KUKA KRL program: pickpallet2.src, pickpallet2.dat

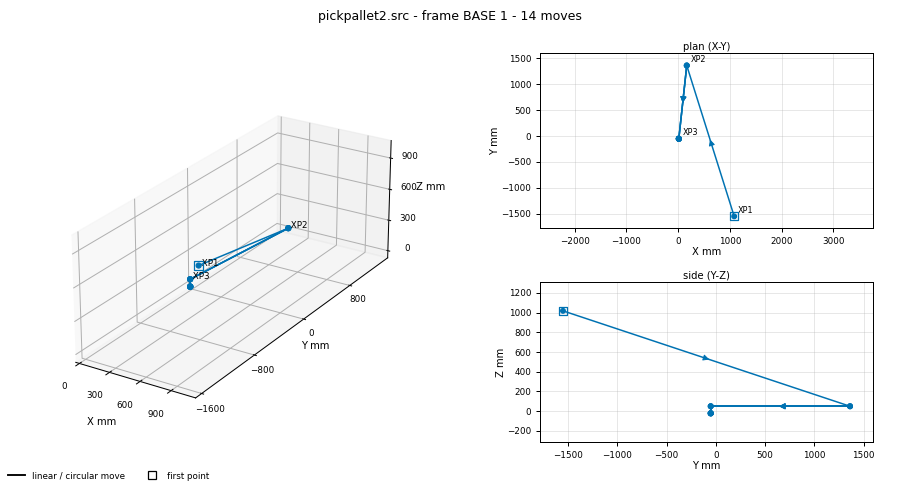
[picture p0: tool path of pickpallet2.src in frame BASE 1, 14 of 20 moves have a stored position in this frame; points joined in program order, loops and branches not executed]
--- pickpallet2.src ---
&ACCESS RVO1
&COMMENT
&ACCESS RVP
&PARAM EDITMASK = *
&PARAM TEMPLATE = C:\KRC\Roboter\Template\vorgabe
&PARAM DISKPATH = KRC:\R1\Program
DEF pickpallet2(pallet1_num:in, Z_pallet:in)
decl pos poz_vz_pal
decl int pallet1_num, ip, Z_pallet
DECL REAL low_z_pallet_pick
decl pos actual_pick_point_1, pallet_pick_point, prp1, prp2, prp9, prp4, prp5

low_z_pallet_pick = 20 ; mm, Z coordinate of the bottom of the first pallet at the pallet pick place

; rotation to the pallet pick place
;FOLD PTP P1  Vel=100 % PDAT1 Tool[2]:tool_empty Base[1]:PickPallet1;%{PE}%R 8.3.22,%MKUKATPBASIS,%CMOVE,%VPTP,%P 1:PTP, 2:P1, 3:, 5:100, 7:PDAT1
$BWDSTART=FALSE
PDAT_ACT=PPDAT1
FDAT_ACT=FP1
BAS(#PTP_PARAMS,100)
PTP XP1
;ENDFOLD

if ((pallet1_num == 10) or (FLAG[5] == FALSE)) then
; movement to the top with search

; rising up
;FOLD LIN P2  Vel=2.00000 m/s CPDAT2 Tool[2]:tool_empty Base[1]:PickPallet1;%{PE}%R 8.3.22,%MKUKATPBASIS,%CMOVE,%VLIN,%P 1:LIN, 2:P2, 3:, 5:2.00000, 7:CPDAT2
$BWDSTART=FALSE
LDAT_ACT=LCPDAT2
FDAT_ACT=FP2
BAS(#CP_PARAMS,2.00000)
LIN XP2
;ENDFOLD

; taking air in order not to avoid the hooks opening
;FOLD SYN OUT 1 'Finger_right'  State= TRUE  at END  Delay= 1500 ms;%{PE}%R 8.3.22,%MKUKATPBASIS,%COUT,%VSYNOUT,%P 2:1, 3:Finger_right, 5:TRUE, 7:1, 9:0, 12:1500
TRIGGER WHEN DISTANCE=1 DELAY=1500 DO $OUT[1]=TRUE
;ENDFOLD
;FOLD SYN OUT 3 'Finger_left'  State= TRUE  at START  Delay= 1500 ms;%{PE}%R 8.3.22,%MKUKATPBASIS,%COUT,%VSYNOUT,%P 2:3, 3:Finger_left, 5:TRUE, 7:0, 9:0, 12:1500
TRIGGER WHEN DISTANCE=0 DELAY=1500 DO $OUT[3]=TRUE
;ENDFOLD

; opening the hooks
;FOLD SYN OUT 5 'All_hooks'  State= TRUE  at END  Delay= 500 ms;%{PE}%R 8.3.22,%MKUKATPBASIS,%COUT,%VSYNOUT,%P 2:5, 3:All_hooks, 5:TRUE, 7:1, 9:0, 12:500
TRIGGER WHEN DISTANCE=1 DELAY=500 DO $OUT[5]=TRUE
;ENDFOLD

; moving to the point above pallet pick place
;FOLD LIN P3  Vel=2.00000 m/s CPDAT3 Tool[2]:tool_empty Base[1]:PickPallet1;%{PE}%R 8.3.22,%MKUKATPBASIS,%CMOVE,%VLIN,%P 1:LIN, 2:P3, 3:, 5:2.00000, 7:CPDAT3
$BWDSTART=FALSE
LDAT_ACT=LCPDAT3
FDAT_ACT=FP3
BAS(#CP_PARAMS,2.00000)
LIN XP3
;ENDFOLD

; stop preprocessor
$ADVANCE = 0

ip = 0
; checking signals from the sensor at the trajectory
INTERRUPT DECL 11 WHEN ((Appr_sensor_signal_1) AND (Appr_sensor_signal_2))  DO STOP (pallet_pick_point, ip)
INTERRUPT ON 11 ; interrupt turn on

; checking signals from the sensor at the trajectory
;FOLD LIN P4  Vel=2.00000 m/s CPDAT4 Tool[2]:tool_empty Base[1]:PickPallet1;%{PE}%R 8.3.22,%MKUKATPBASIS,%CMOVE,%VLIN,%P 1:LIN, 2:P4, 3:, 5:2.00000, 7:CPDAT4
$BWDSTART=FALSE
LDAT_ACT=LCPDAT4
FDAT_ACT=FP4
BAS(#CP_PARAMS,2.00000)
LIN XP4
;ENDFOLD

; interrupt turn off
INTERRUPT OFF 11

IF ip == 1 THEN
pallet_pick_point.z = pallet_pick_point.z - 20 ; if pallet was found than pulling down to if after the event when the sensor had found it
ELSE
pallet_pick_point = XP4
ENDIF

pallet1_num = (low_z_pallet_pick + pallet_pick_point.z) / Z_pallet ; calculation of number of pallets

; sinking to the pick point
;FOLD LIN pallet_pick_point  Vel=2.00000 m/s CPDAT4 Tool[2]:tool_empty Base[1]:PickPallet1;%{PE}%R 8.3.22,%MKUKATPBASIS,%CMOVE,%VLIN,%P 1:LIN, 2:pallet_pick_point, 3:, 5:2.00000, 7:CPDAT4
$BWDSTART=FALSE
LDAT_ACT=LCPDAT4
FDAT_ACT=FP4
BAS(#CP_PARAMS,2.00000)
LIN Xpallet_pick_point
;ENDFOLD

; movement relative to the actual_pick_point_1 to the defined length down
;FOLD OUT 5 'all hooks'  State= FALSE;%{PE}%R 8.3.22,%MKUKATPBASIS,%COUT,%VOUTX,%P 2:5, 3:all hooks, 5:FALSE, 6:

$OUT[5]=FALSE
;ENDFOLD

; start preprocessor
$ADVANCE = 3

prp1 = pallet_pick_point
prp1.z = prp1.z + 200 ; rising up to the defined length

;FOLD LIN prp1 CONT Vel=2.00000 m/s CPDAT5 Tool[4]:tool_pallet Base[1]:PickPallet1;%{PE}%R 8.3.22,%MKUKATPBASIS,%CMOVE,%VLIN,%P 1:LIN, 2:prp1, 3:C_DIS C_DIS, 5:2.00000, 7:CPDAT5
$BWDSTART=FALSE
LDAT_ACT=LCPDAT5
FDAT_ACT=Fprp1
BAS(#CP_PARAMS,2.00000)
LIN Xprp1 C_DIS C_DIS
;ENDFOLD

;calculation of the coordinates of the retreat points
XP5.z = pallet_pick_point.z
XP6.z = pallet_pick_point.z

; retreat to the approach points
;FOLD LIN P5 CONT Vel=2.00000 m/s CPDAT5 Tool[4]:tool_pallet Base[1]:PickPallet1;%{PE}%R 8.3.22,%MKUKATPBASIS,%CMOVE,%VLIN,%P 1:LIN, 2:P5, 3:C_DIS C_DIS, 5:2.00000, 7:CPDAT5
$BWDSTART=FALSE
LDAT_ACT=LCPDAT5
FDAT_ACT=FP5
BAS(#CP_PARAMS,2.00000)
LIN XP5 C_DIS C_DIS
;ENDFOLD
;FOLD PTP P6 CONT Vel=100 % PDAT6 Tool[4]:tool_pallet Base[1]:PickPallet1;%{PE}%R 8.3.22,%MKUKATPBASIS,%CMOVE,%VPTP,%P 1:PTP, 2:P6, 3:C_PTP, 5:100, 7:PDAT6
$BWDSTART=FALSE
PDAT_ACT=PPDAT6
FDAT_ACT=FP6
BAS(#PTP_PARAMS,100)
PTP XP6 C_PTP
;ENDFOLD



ELSE
if ((pallet1_num > 5) and (FLAG[5] == TRUE)) then
; movement along the calculated coordinateswithout search along the upper trajectory

; rising up
;FOLD LIN P2  Vel=2.00000 m/s CPDAT2 Tool[2]:tool_empty Base[1]:PickPallet1;%{PE}%R 8.3.22,%MKUKATPBASIS,%CMOVE,%VLIN,%P 1:LIN, 2:P2, 3:, 5:2.00000, 7:CPDAT2
$BWDSTART=FALSE
LDAT_ACT=LCPDAT2
FDAT_ACT=FP2
BAS(#CP_PARAMS,2.00000)
LIN XP2
;ENDFOLD

; taking air in order not to avoid the hooks opening
;FOLD SYN OUT 1 'Finger_right'  State= TRUE  at END  Delay= 1500 ms;%{PE}%R 8.3.22,%MKUKATPBASIS,%COUT,%VSYNOUT,%P 2:1, 3:Finger_right, 5:TRUE, 7:1, 9:0, 12:1500
TRIGGER WHEN DISTANCE=1 DELAY=1500 DO $OUT[1]=TRUE
;ENDFOLD
;FOLD SYN OUT 3 'Finger_left'  State= TRUE  at START  Delay= 1500 ms;%{PE}%R 8.3.22,%MKUKATPBASIS,%COUT,%VSYNOUT,%P 2:3, 3:Finger_left, 5:TRUE, 7:0, 9:0, 12:1500
TRIGGER WHEN DISTANCE=0 DELAY=1500 DO $OUT[3]=TRUE
;ENDFOLD

; opening the hooks
;FOLD SYN OUT 5 'All_hooks'  State= TRUE  at END  Delay= 500 ms;%{PE}%R 8.3.22,%MKUKATPBASIS,%COUT,%VSYNOUT,%P 2:5, 3:All_hooks, 5:TRUE, 7:1, 9:0, 12:500
TRIGGER WHEN DISTANCE=1 DELAY=500 DO $OUT[5]=TRUE
;ENDFOLD

; moving to the point above pallet pick place
;FOLD LIN P3  Vel=2.00000 m/s CPDAT3 Tool[2]:tool_empty Base[1]:PickPallet1;%{PE}%R 8.3.22,%MKUKATPBASIS,%CMOVE,%VLIN,%P 1:LIN, 2:P3, 3:, 5:2.00000, 7:CPDAT3
$BWDSTART=FALSE
LDAT_ACT=LCPDAT3
FDAT_ACT=FP3
BAS(#CP_PARAMS,2.00000)
LIN XP3
;ENDFOLD

pallet_pick_point = XP4
pallet_pick_point.z = pallet1_num * Z_pallet - low_z_pallet_pick ; calculation of the pick point coordinates according to number of pallets

; sinking to the pick point
;FOLD LIN pallet_pick_point  Vel=2.00000 m/s CPDAT4 Tool[2]:tool_empty Base[1]:PickPallet1;%{PE}%R 8.3.22,%MKUKATPBASIS,%CMOVE,%VLIN,%P 1:LIN, 2:pallet_pick_point, 3:, 5:2.00000, 7:CPDAT4
$BWDSTART=FALSE
LDAT_ACT=LCPDAT4
FDAT_ACT=FP4
BAS(#CP_PARAMS,2.00000)
LIN Xpallet_pick_point
;ENDFOLD

; movement relative to the actual_pick_point_1 to the defined length down
;FOLD OUT 5 'all hooks'  State= FALSE;%{PE}%R 8.3.22,%MKUKATPBASIS,%COUT,%VOUTX,%P 2:5, 3:all hooks, 5:FALSE, 6:

$OUT[5]=FALSE
;ENDFOLD

prp1 = pallet_pick_point
prp1.z = prp1.z + 200 ; rising up to the defined length

;FOLD LIN prp1 CONT Vel=2.00000 m/s CPDAT5 Tool[4]:tool_pallet Base[1]:PickPallet1;%{PE}%R 8.3.22,%MKUKATPBASIS,%CMOVE,%VLIN,%P 1:LIN, 2:prp1, 3:C_DIS C_DIS, 5:2.00000, 7:CPDAT5
$BWDSTART=FALSE
LDAT_ACT=LCPDAT5
FDAT_ACT=Fprp1
BAS(#CP_PARAMS,2.00000)
LIN Xprp1 C_DIS C_DIS
;ENDFOLD

;calculation of the coordinates of the retreat points
XP5.z = pallet_pick_point.z
XP6.z = pallet_pick_point.z

; retreat to the approach points
;FOLD LIN P5 CONT Vel=2.00000 m/s CPDAT5 Tool[4]:tool_pallet Base[1]:PickPallet1;%{PE}%R 8.3.22,%MKUKATPBASIS,%CMOVE,%VLIN,%P 1:LIN, 2:P5, 3:C_DIS C_DIS, 5:2.00000, 7:CPDAT5
$BWDSTART=FALSE
LDAT_ACT=LCPDAT5
FDAT_ACT=FP5
BAS(#CP_PARAMS,2.00000)
LIN XP5 C_DIS C_DIS
;ENDFOLD
;FOLD PTP P6 CONT Vel=100 % PDAT6 Tool[4]:tool_pallet Base[1]:PickPallet1;%{PE}%R 8.3.22,%MKUKATPBASIS,%CMOVE,%VPTP,%P 1:PTP, 2:P6, 3:C_PTP, 5:100, 7:PDAT6
$BWDSTART=FALSE
PDAT_ACT=PPDAT6
FDAT_ACT=FP6
BAS(#PTP_PARAMS,100)
PTP XP6 C_PTP
;ENDFOLD



Else
If ((pallet1_num < 5) and (FLAG[5]== TRUE)) then
; movement along the calculated coordinateswithout search along the lower trajectory

prp2 = XP2
prp3 = XP3
prp2.z = prp2.z - 200
prp3.z = prp3.z - 200


; rising up
;FOLD LIN prp2  Vel=2.00000 m/s CPDAT2 Tool[2]:tool_empty Base[1]:PickPallet1;%{PE}%R 8.3.22,%MKUKATPBASIS,%CMOVE,%VLIN,%P 1:LIN, 2:prp2, 3:, 5:2.00000, 7:CPDAT2
$BWDSTART=FALSE
LDAT_ACT=LCPDAT2
FDAT_ACT=FP2
BAS(#CP_PARAMS,2.00000)
LIN Xprp2
;ENDFOLD

; taking air in order not to avoid the hooks opening
;FOLD SYN OUT 1 'Finger_right'  State= TRUE  at END  Delay= 1500 ms;%{PE}%R 8.3.22,%MKUKATPBASIS,%COUT,%VSYNOUT,%P 2:1, 3:Finger_right, 5:TRUE, 7:1, 9:0, 12:1500
TRIGGER WHEN DISTANCE=1 DELAY=1500 DO $OUT[1]=TRUE
;ENDFOLD
;FOLD SYN OUT 3 'Finger_left'  State= TRUE  at START  Delay= 1500 ms;%{PE}%R 8.3.22,%MKUKATPBASIS,%COUT,%VSYNOUT,%P 2:3, 3:Finger_left, 5:TRUE, 7:0, 9:0, 12:1500
TRIGGER WHEN DISTANCE=0 DELAY=1500 DO $OUT[3]=TRUE
;ENDFOLD

; opening the hooks
;FOLD SYN OUT 5 'All_hooks'  State= TRUE  at END  Delay= 500 ms;%{PE}%R 8.3.22,%MKUKATPBASIS,%COUT,%VSYNOUT,%P 2:5, 3:All_hooks, 5:TRUE, 7:1, 9:0, 12:500
TRIGGER WHEN DISTANCE=1 DELAY=500 DO $OUT[5]=TRUE
;ENDFOLD

; moving to the point above pallet pick place
;FOLD LIN prp3  Vel=2.00000 m/s CPDAT3 Tool[2]:tool_empty Base[1]:PickPallet1;%{PE}%R 8.3.22,%MKUKATPBASIS,%CMOVE,%VLIN,%P 1:LIN, 2:prp3, 3:, 5:2.00000, 7:CPDAT3
$BWDSTART=FALSE
LDAT_ACT=LCPDAT3
FDAT_ACT=Fp3
BAS(#CP_PARAMS,2.00000)
LIN Xprp3
;ENDFOLD

pallet_pick_point = XP4
pallet_pick_point.z = pallet1_num * Z_pallet - low_z_pallet_pick ; calculation of the pick point coordinates according to number of pallets

; sinking to the pick point
;FOLD LIN pallet_pick_point  Vel=2.00000 m/s CPDAT4 Tool[2]:tool_empty Base[1]:PickPallet1;%{PE}%R 8.3.22,%MKUKATPBASIS,%CMOVE,%VLIN,%P 1:LIN, 2:pallet_pick_point, 3:, 5:2.00000, 7:CPDAT4
$BWDSTART=FALSE
LDAT_ACT=LCPDAT4
FDAT_ACT=FP4
BAS(#CP_PARAMS,2.00000)
LIN Xpallet_pick_point
;ENDFOLD

; movement relative to the actual_pick_point_1 to the defined length down
;FOLD OUT 5 'all hooks'  State= FALSE;%{PE}%R 8.3.22,%MKUKATPBASIS,%COUT,%VOUTX,%P 2:5, 3:all hooks, 5:FALSE, 6:

$OUT[5]=FALSE
;ENDFOLD

prp1 = pallet_pick_point
prp1.z = prp1.z + 200 ; rising up to the defined length

;FOLD LIN prp1 CONT Vel=2.00000 m/s CPDAT5 Tool[4]:tool_pallet Base[1]:PickPallet1;%{PE}%R 8.3.22,%MKUKATPBASIS,%CMOVE,%VLIN,%P 1:LIN, 2:prp1, 3:C_DIS C_DIS, 5:2.00000, 7:CPDAT5
$BWDSTART=FALSE
LDAT_ACT=LCPDAT5
FDAT_ACT=Fprp1
BAS(#CP_PARAMS,2.00000)
LIN Xprp1 C_DIS C_DIS
;ENDFOLD

;calculation of the coordinates of the retreat points
XP5.z = pallet_pick_point.z
XP6.z = pallet_pick_point.z

; retreat to the approach points
;FOLD LIN P5 CONT Vel=2.00000 m/s CPDAT5 Tool[4]:tool_pallet Base[1]:PickPallet1;%{PE}%R 8.3.22,%MKUKATPBASIS,%CMOVE,%VLIN,%P 1:LIN, 2:P5, 3:C_DIS C_DIS, 5:2.00000, 7:CPDAT5
$BWDSTART=FALSE
LDAT_ACT=LCPDAT5
FDAT_ACT=FP5
BAS(#CP_PARAMS,2.00000)
LIN XP5 C_DIS C_DIS
;ENDFOLD
;FOLD PTP P6 CONT Vel=100 % PDAT6 Tool[4]:tool_pallet Base[1]:PickPallet1;%{PE}%R 8.3.22,%MKUKATPBASIS,%CMOVE,%VPTP,%P 1:PTP, 2:P6, 3:C_PTP, 5:100, 7:PDAT6
$BWDSTART=FALSE
PDAT_ACT=PPDAT6
FDAT_ACT=FP6
BAS(#PTP_PARAMS,100)
PTP XP6 C_PTP
;ENDFOLD

ENDIF
ENDIF
ENDIF

END

--- pickpallet2.dat ---
DEFDAT pickpallet2 PUBLIC
;FOLD EXTERNAL DECLARATIONS;%{PE}%MKUKATPBASIS,%CEXT,%VCOMMON,%P
;FOLD BASISTECH EXT;%{PE}%MKUKATPBASIS,%CEXT,%VEXT,%P
EXT  BAS (BAS_COMMAND  :IN,REAL  :IN )
DECL INT SUCCESS
;ENDFOLD (BASISTECH EXT)
;FOLD USER EXT;%{E}%MKUKATPUSER,%CEXT,%VEXT,%P
;Make your modifications here

;ENDFOLD (USER EXT)
;ENDFOLD (EXTERNAL DECLARATIONS)
; DECL BASIS_SUGG_T LAST_BASIS={POINT1[] "P15                     ",POINT2[] "P15                     ",CP_PARAMS[] "CPDAT15                 ",PTP_PARAMS[] "PDAT4                   ",CONT[] "                        ",CP_VEL[] "2                       ",PTP_VEL[] "100                     ",SYNC_PARAMS[] "SYNCDAT                 ",SPL_NAME[] "S0                      ",A_PARAMS[] "ADAT0                   "}
DECL E6POS XP1={X 1082.92773,Y -1551.50513,Z 1017.75269,A 1.30770361,B -3.12852907E-14,C -180.000,S 2,T 3,E1 0.0,E2 0.0,E3 0.0,E4 0.0,E5 0.0,E6 0.0}
DECL FDAT FP1={TOOL_NO 2,BASE_NO 1,IPO_FRAME #BASE,POINT2[] " ",TQ_STATE FALSE}
DECL PDAT PPDAT1={VEL Vel_without_load_ptp,ACC 100,APO_DIST 100,APO_MODE #CPTP,GEAR_JERK 50}

DECL E6POS XP2={X 166.779327,Y 1361.41699,Z 49.6159210,A 2.20242882,B 3.19880265E-14,C 180.000,S 2,T 3,E1 0.0,E2 0.0,E3 0.0,E4 0.0,E5 0.0,E6 0.0}
DECL FDAT FP2={TOOL_NO 2,BASE_NO 1,IPO_FRAME #BASE,POINT2[] " ",TQ_STATE FALSE}
DECL LDAT LCPDAT2={VEL 2.00000,ACC 100,APO_DIST 100,APO_FAC 50,AXIS_VEL 100.0,AXIS_ACC 100.0,ORI_TYP #VAR,CIRC_TYP #BASE,JERK_FAC 50.0,GEAR_JERK 50.0,EXAX_IGN 0}

DECL E6POS XP3={X 13.2864075,Y -52.1582222,Z 49.6159210,A 2.20242858,B 3.91124367E-15,C 180.000,S 2,T 3,E1 0.0,E2 0.0,E3 0.0,E4 0.0,E5 0.0,E6 0.0}
DECL FDAT FP3={TOOL_NO 2,BASE_NO 1,IPO_FRAME #BASE,POINT2[] " ",TQ_STATE FALSE}
DECL LDAT LCPDAT3={VEL 2.00000,ACC 100,APO_DIST 100,APO_FAC 50,AXIS_VEL 100.0,AXIS_ACC 100.0,ORI_TYP #VAR,CIRC_TYP #BASE,JERK_FAC 50.0,GEAR_JERK 50.0,EXAX_IGN 0}

DECL E6POS XP4={X 13.2864075,Y -52.1582222,Z -21.7196426,A 2.20242858,B 3.91124367E-15,C 180.000,S 2,T 3,E1 0.0,E2 0.0,E3 0.0,E4 0.0,E5 0.0,E6 0.0}
DECL FDAT FP4={TOOL_NO 2,BASE_NO 1,IPO_FRAME #BASE,POINT2[] " ",TQ_STATE FALSE}
DECL LDAT LCPDAT4={VEL 2.00000,ACC 100,APO_DIST 100,APO_FAC 50,AXIS_VEL 100.0,AXIS_ACC 100.0,ORI_TYP #VAR,CIRC_TYP #BASE,JERK_FAC 50.0,GEAR_JERK 50.0,EXAX_IGN 0}

DECL E6POS XP5={X 13.2864075,Y -52.1582222,Z 860.575439,A 2.20242858,B 1.14588489E-14,C 180.000,S 2,T 3,E1 0.0,E2 0.0,E3 0.0,E4 0.0,E5 0.0,E6 0.0}
DECL FDAT FP5={TOOL_NO 4,BASE_NO 1,IPO_FRAME #BASE,POINT2[] " ",TQ_STATE FALSE}
DECL LDAT LCPDAT5={VEL 2.00000,ACC 100,APO_DIST 100,APO_FAC 50,AXIS_VEL 100.0,AXIS_ACC 100.0,ORI_TYP #VAR,CIRC_TYP #BASE,JERK_FAC 50.0,GEAR_JERK 50.0,EXAX_IGN 0}

DECL E6POS XP6={X 166.779327,Y 1361.41699,Z 49.6159210,A 2.20242882,B 3.19880265E-14,C 180.000,S 2,T 3,E1 0.0,E2 0.0,E3 0.0,E4 0.0,E5 0.0,E6 0.0}
DECL FDAT FP6={TOOL_NO 4,BASE_NO 1,IPO_FRAME #BASE,POINT2[] " ",TQ_STATE FALSE}
DECL PDAT PPDAT6={VEL 100,ACC 100,APO_DIST 100,APO_MODE #CPTP,GEAR_JERK 50}

DECL E6POS Xpallet_pick_point={X 13.2864075,Y -52.1582222,Z -21.7196426,A 2.20242858,B 3.91124367E-15,C 180.000,S 2,T 3,E1 0.0,E2 0.0,E3 0.0,E4 0.0,E5 0.0,E6 0.0}
DECL FDAT Fpallet_pick_point={TOOL_NO 2,BASE_NO 1,IPO_FRAME #BASE,POINT2[] " ",TQ_STATE FALSE}

DECL E6POS Xprp1={X 13.2864075,Y -52.1582222,Z -21.7196426,A 2.20242858,B 3.91124367E-15,C 180.000,S 2,T 3,E1 0.0,E2 0.0,E3 0.0,E4 0.0,E5 0.0,E6 0.0}
DECL FDAT Fprp1={TOOL_NO 4,BASE_NO 1,IPO_FRAME #BASE,POINT2[] " ",TQ_STATE FALSE}

DECL E6POS Xprp2={X 166.779327,Y 1361.41699,Z 49.6159210,A 2.20242882,B 3.19880265E-14,C 180.000,S 2,T 3,E1 0.0,E2 0.0,E3 0.0,E4 0.0,E5 0.0,E6 0.0}
DECL FDAT Fprp2={TOOL_NO 2,BASE_NO 1,IPO_FRAME #BASE,POINT2[] " ",TQ_STATE FALSE}

DECL E6POS Xprp3={X 13.2864075,Y -52.1582222,Z 49.6159210,A 2.20242858,B 3.91124367E-15,C 180.000,S 2,T 3,E1 0.0,E2 0.0,E3 0.0,E4 0.0,E5 0.0,E6 0.0}
DECL FDAT Fprp3={TOOL_NO 2,BASE_NO 1,IPO_FRAME #BASE,POINT2[] " ",TQ_STATE FALSE}
ENDDAT
